(* IEC 61131-3 sources: HydroSim/openplc, 1 file *)

(* ---- script.st ---- *)
PROGRAM PLC_PRG
VAR
    x : BOOL := TRUE;
END_VAR

END_PROGRAM
